Staubli VAL3: OnF1.pgx

public program OnF1()
begin
  taskCreate "Motion",100,SingleMotion(sPath,true,0)
  wait(taskStatus("Motion")==1)
end
